// SIMATIC S7-200 project (STEP 7-Micro/WIN), CPU 224XP CN REL 02.01

ORGANIZATION_BLOCK 程序块:OB1
TITLE=项目信息
// 这个PLC程序实现了S7-200 PLC与LG变频器的Modbus通信
// S7-200作为Modbus主站，软件版本必须升级到SP5,即桌面显示：V4.0 STEP 7 MicroWIN SP5
// 如果你的版本是SP4以下的，那么只能作为Modbus丛站，
// 下载SP5的地方可到【西门子常规软件下载】
// http://xmz.ymmfa.com  中的论坛下载。
// 设备信息
// 系统涉及的物理设备包括S7-200 PLC和LG变频器。
// 系统实现
// 系统启动时，首先初始化Modbus通信，波特率为19200，无奇偶校验，超时时间为1000ms，确保与变频器的通信参数匹配。通信初始化完成后，系统进入通信就绪状态。
// 当操作员按下正向起动按钮时，系统检查反向起动按钮和停止按钮是否未激活。只有在这些条件满足时，系统启动电机正向运行，传送带开始向前移动。同时，一个定时器启动，计时后结束本次操作。
// 类似地，当操作员按下反向起动按钮时，系统确认正向起动按钮和停止按钮未激活后，启动电机反向运行，传送带向后移动。另一个定时器计时后完成操作。
// 若操作员按下停止按钮，系统检查反向起动按钮和另一操作未激活后，停止电机运行，传送带静止。一个定时器计时后复位停止状态。
// 在发送Modbus请求前，系统确保正向起动、反向起动和停止操作均未激活，只有在此情况下更新控制参数并设置目标地址，避免操作冲突。正向起动、反向起动和停止操作通过条件检查实现互斥，确保电机运行状态清晰和安全。
BEGIN
Network 1
LD     SM0.0
=      L60.0
LD     SM0.0
=      L63.7
LD     L60.0
CALL   MBUS_CTRL:SBR1, L63.7, 19200, 0, 1000, M20.2, VB502
Network 2
LD     T36
=      M2.6
S      M2.7, 1
Network 3
LDN    M2.3
AN     M2.1
AN     M2.2
MOVW   VW680, VW660
MOVD   40006, VD602
Network 4
// MBUS_MSG指令(或用于端口1的MBUS_MSG_P1)用于启动对Modbus从站的请求并处理应答。
// First："首次"参数应该在有新请求要发送时才打开以进行一次扫描。"首次"输入应当通过一个边沿检测元素(例如               上升沿)打开，这将导致请求被传送一次。参见实例程序。
// Slave："从站"参数是Modbus从站的地址。允许的范围是0到247。地址0是广播地址，只能用于写请求。不存在对             地址0的广播请求的应答。并非所有的从站会支持广播地址。S7-200 Modbus从站协议库不支持广播地址。
//            此处值＝1，表示对1号丛站进行读写
// RW："读写"参出指定是否要读取或写入该消息。"读写"参数允许使用下列两个值。
// 
//              0 � 读
//              1 � 写
// Addr："地址"参数是起始的Modbus地址。允许使用下列取值范围：00001至09999是离散输出(线圈)
// 
//            10001至19999是离散输入(触点)
//            30001至39999是输入寄存器
//            40001至49999是保持寄存器
//            "地址"的指定取值范围基于Modbus从站支持的地址。
// Count："计数"参数指定在该请求中读取或写入的数据元素的数目。"计数"值是位数(对于位数据类型)和字数(对于字数据类型)。
// 
//              地址0xxxx � "计数"是要读取或写入的位数。
//              地址1xxxx � "计数"是要读取的位数。
//              地址3xxxx � "计数"是要读取的输入寄存器的字数。
//              地址4xxxx � "计数"是要读取或写入的保持寄存器的字数。
// 
// MBUS_MSG指令将读取或写入最大120个字或1920个位(240字节的数据)。"计数"的实际限值将取决于Modbus从站中的限制。
// 
// DataPtr："DataPtr"参数是指向S7-200 CPU的V存储器中与读取或写入请求相关的数据的间接地址指针。对于读取请求，DataPtr应该指向用于存储从Modbus从站读取的数据的第一个CPU存储器位置。对于写入请求，DataPtr应该指向要发送到Modbus从站的数据的第一个CPU存储器位置。
// DataPtr值作为间接地址指针传递到MBUS_MSG。
// 
LD     SM0.0
=      L60.0
LD     SM0.0
=      L63.7
LD     L60.0
CALL   MBUS_MSG:SBR2, L63.7, 1, 1, VD602, 1, &VB600, M20.1, VB506
Network 5
LD     SM0.0
MOVW   VW660, VW600
Network 6
// 正向起动
LD     M20.6
AN     M21.1
AN     M21.2
EU
S      M2.1, 1
Network 7
// 正向起动
LD     M2.1
LPS
MOVW   16#2, VW660
MOVD   40007, VD602
TON    T33, 200
ED
TOF    T36, 500
LPP
A      T33
R      M2.1, 1
Network 8
// 反向起动
LD     M21.1
AN     M20.6
AN     M21.2
EU
S      M2.2, 1
Network 9
// 反向起动
LD     M2.2
LPS
AN     SM0.5
MOVW   16#4, VW660
LRD
AN     SM0.5
MOVD   40007, VD602
LRD
TON    T34, 200
LPP
A      T34
R      M2.2, 1
Network 10
// 停止
LD     M21.2
AN     M21.1
AN     M21.6
EU
S      M2.3, 1
Network 11
// 停止
LD     M2.3
LPS
AN     SM0.5
MOVW   16#0, VW660
LRD
AN     SM0.5
MOVD   40007, VD602
LRD
TON    T35, 300
LPP
A      T35
R      M2.3, 1
END_ORGANIZATION_BLOCK

// SBR1: protected block, not included

// SBR2: protected block, not included

// SBR3: protected block, not included
